(* PLC project Test Library, INSA Strasbourg Test Library 1.0, author Mathieu Giamberini *)
(* stored: creationDateTime 2024-10-04T15:34:52, modificationDateTime 2024-10-04T15:56:57 *)

(* This block outputs the sum of input I0 and 10. *)
FUNCTION_BLOCK Test
  VAR_INPUT
    I0 : INT;  (* Insert an integer here *)
    ACTIVE : BOOL;  (* 0 - block does nothing, 1 - block sums 10 to integer in I0 *)
  END_VAR
  VAR_OUTPUT
    OUT : INT;  (* This is the output: I0 + 10 *)
  END_VAR

            IF ACTIVE = TRUE T HEN
OUT := I0 + 10;
END_IF;
          
END_FUNCTION_BLOCK

(* This block ouput the chip id (0xA0) and 0xFF for error *)
FUNCTION_BLOCK BNO055
  VAR_OUTPUT
    CHIP_ID : BYTE;  (* Chip id : 0xA0 *)
  END_VAR

            
CHIP_ID := 0xFF;

          
END_FUNCTION_BLOCK
